// TIA Portal V21 export
// export: Created 2026-08-26T08:42:39.6370071Z, ExportSetting None, DisplayName Totally Integrated Automation Portal, DisplayVersion V21, DisplayName STEP 7 Professional, DisplayVersion V21, DisplayName STEP 7 Safety, DisplayVersion V21, DisplayName Tech WebApplication, DisplayVersion V21, DisplayName WinCC Basic/Comfort/Advanced, DisplayVersion V21
FUNCTION_BLOCK "TASK012A_FB_Callee"   // FB1, LAD
{ S7_Optimized_Access := 'TRUE' }
// stored: MemoryReserve 100, SetENOAutomatically false
   VAR_INPUT
      Enable : Bool;
   END_VAR
   VAR_OUTPUT
      Active : Bool;
   END_VAR
BEGIN

REGION Network 1
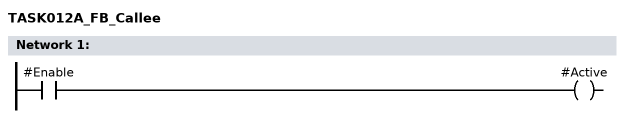
   RUNG wire#powerrail
      Contact( #Enable )
      Coil( #Active )
   END_RUNG
   // the same network as SCL:
   #Active := #Enable;
END_REGION
END_FUNCTION_BLOCK
